KUKA KRL program: Rack_Verde_Cerrar_D.src, Rack_Verde_Cerrar_D.dat

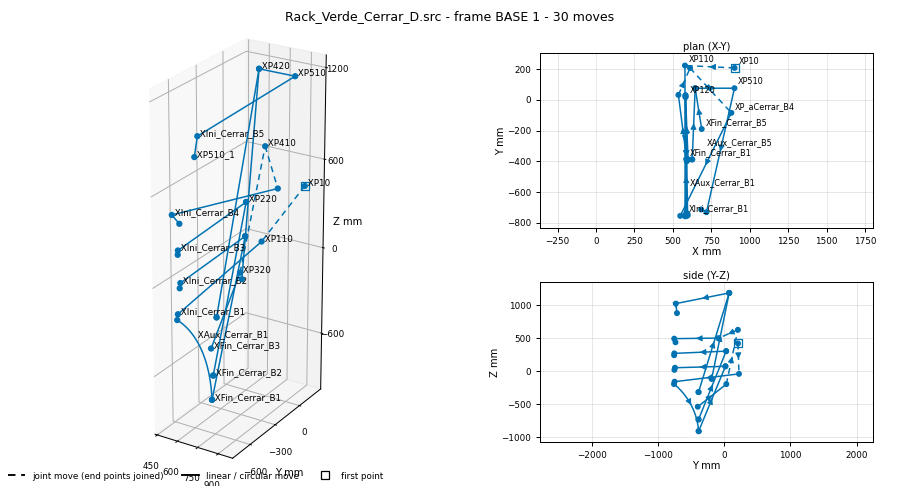
[picture p0: tool path of Rack_Verde_Cerrar_D.src in frame BASE 1, 30 of 38 moves have a stored position in this frame; points joined in program order, loops and branches not executed]
--- Rack_Verde_Cerrar_D.src ---
&ACCESS RVO1
&REL 165
&COMMENT CERRAR BANDEJAS PRG
&PARAM EDITMASK = *
&PARAM TEMPLATE = C:\KRC\Roboter\Template\vorgabe
&PARAM DISKPATH = KRC:\R1\Program\MAFELEC
DEF Rack_Verde_Cerrar_D( )
;FOLD INI;%{PE}
  ;FOLD BASISTECH INI
    GLOBAL INTERRUPT DECL 3 WHEN $STOPMESS==TRUE DO IR_STOPM ( )
    INTERRUPT ON 3
    BAS (#INITMOV,0 )
  ;ENDFOLD (BASISTECH INI)
;FOLD SPOTTECH INI
USERSPOT(#INIT)
;ENDFOLD (SPOTTECH INI)
;FOLD GRIPPERTECH INI
USER_GRP(0,DUMMY,DUMMY,GDEFAULT)
;ENDFOLD (GRIPPERTECH INI)
  ;FOLD USER INI
    ;Make your modifications here
INTERRUPT DECL 81 WHEN I_121R1S501 DO STOP_PUSH()
INTERRUPT DECL 91 WHEN I_121R1S502 DO STOP_PUSH()

O_TYPE_INFO=0

  ;ENDFOLD (USER INI)
;ENDFOLD (INI)
;################################################
; PROYECTO: MAFELEC PLANTA DE BATERIAS
; ROBOT: 121_R1
; PROGRAMA: CERRAR BANDEJAS EN RACK VERDE
; CREADO POR: Alejandro Company(zaisor robotics)
; FECHA: 23-NOVIEMBRE-2022
; MODIFICADO POR:
; FECHA MODIFICACION: 20-ENERO-2023
;################################################

$TIMER[5]=0
$TIMER_STOP[5]=FALSE

PTP $POS_ACT
Empujador(1,"A",FALSE)
Empujador(2,"R",FALSE)

;FOLD BORRADO SEÑALES INPICKER
O_INPICKER_OK=FALSE
O_INPICKER_NOK=FALSE
O_LIMITS_OK=FALSE
O_LIMITS_NOK=FALSE
O_LIMIT_X=FALSE
O_LIMIT_Y=FALSE
O_LIMIT_Z=FALSE
O_LIMIT_A=FALSE
O_LIMIT_B=FALSE
O_LIMIT_C=FALSE
;ENDFOLD

;INTERRUPT ON 81

INI_BUCLE:
;FOLD LIN P10 Vel=0.05 m/s M Tool[1]:T_PUSH1 Base[1]:Rack_Verde;%{PE}%R 8.3.48,%MKUKATPBASIS,%CMOVE,%VLIN,%P 1:LIN, 2:P10, 3:, 5:0.05, 7:M
$BWDSTART=FALSE
LDAT_ACT=LM
FDAT_ACT=FP10
BAS(#CP_PARAMS,0.05)
LIN XP10
;ENDFOLD

If ($SR_RANGE_ACTIVE[16]==FALSE) THEN
$out[61]=TRUE
WAIT FOR FALSE
WAIT FOR FALSE
WAIT FOR FALSE
;SETA DE BOMBEROS PULSADA, LLEVAR ROBOT A HOME Y REINICIAR PROGRAMA PARA RESTABLECER
ENDIF


WAIT FOR I_121R1S1000==FALSE
Empujador(1,"A",TRUE)
Empujador(2,"R",TRUE)
$ADVANCE=0

WAIT FOR (RV_Bandeja_Nr>10) AND (RV_Bandeja_Nr<16)

;PETICION CLAUSURA BANDEJAS EN RACK VERDE
SWITCH RV_Bandeja_Nr ;

CASE 11
O_TYPE_RQ=FALSE
O_TYPE_INFO=RV_Bandeja_Nr

;FOLD PTP P110 CONT Vel=50 % M Tool[1]:T_PUSH1 Base[1]:Rack_Verde;%{PE}%R 8.3.48,%MKUKATPBASIS,%CMOVE,%VPTP,%P 1:PTP, 2:P110, 3:C_DIS, 5:50, 7:M
$BWDSTART=FALSE
PDAT_ACT=PM
FDAT_ACT=FP110
BAS(#PTP_PARAMS,50)
PTP XP110 C_DIS
;ENDFOLD

WAIT FOR I_RackVerde_Pin1A
WAIT FOR I_Rack1_S1==TRUE
O_TREQ_2=TRUE

;FOLD LIN Ini_Cerrar_B1 Vel=1 m/s M Tool[1]:T_PUSH1 Base[1]:Rack_Verde;%{PE}%R 8.3.48,%MKUKATPBASIS,%CMOVE,%VLIN,%P 1:LIN, 2:Ini_Cerrar_B1, 3:, 5:1, 7:M
$BWDSTART=FALSE
LDAT_ACT=LM
FDAT_ACT=FIni_Cerrar_B1
BAS(#CP_PARAMS,1)
LIN XIni_Cerrar_B1
;ENDFOLD
;FOLD LIN P110_1 Vel=1 m/s M Tool[1]:T_PUSH1 Base[1]:Rack_Verde;%{PE}%R 8.3.48,%MKUKATPBASIS,%CMOVE,%VLIN,%P 1:LIN, 2:P110_1, 3:, 5:1, 7:M
$BWDSTART=FALSE
LDAT_ACT=LM
FDAT_ACT=FP110_1
BAS(#CP_PARAMS,1)
LIN XP110_1
;ENDFOLD

O_TREQ_2=TRUE
WAIT FOR I_TRDY_2
O_TREQ_2=FALSE

;FOLD CIRC Aux_Cerrar_B1 Fin_Cerrar_B1 Vel=1 m/s M Tool[1]:T_PUSH1 Base[1]:Rack_Verde;%{PE}%R 8.3.48,%MKUKATPBASIS,%CMOVE,%VCIRC,%P 1:CIRC, 2:Aux_Cerrar_B1, 3:Fin_Cerrar_B1, 4:, 6:1, 8:M
$BWDSTART=FALSE
LDAT_ACT=LM
FDAT_ACT=FFin_Cerrar_B1
BAS(#CP_PARAMS,1)
CIRC XAux_Cerrar_B1, XFin_Cerrar_B1
;ENDFOLD
;FOLD LIN Fin_Cerrar_B1 Vel=0.5 m/s CPDAT2 Tool[1]:T_PUSH1 Base[1]:Rack_Verde;%{PE}%R 8.3.48,%MKUKATPBASIS,%CMOVE,%VLIN,%P 1:LIN, 2:Fin_Cerrar_B1, 3:, 5:0.5, 7:CPDAT2
$BWDSTART=FALSE
LDAT_ACT=LCPDAT2
FDAT_ACT=FFin_Cerrar_B1
BAS(#CP_PARAMS,0.5)
LIN XFin_Cerrar_B1
;ENDFOLD
IF ($IN[64]==TRUE) THEN
;FOLD MOVIMIENTO CONTROLADO CERRAR BANDEJA

   $OUT[63]=TRUE ; DESHABILITAMOS EL CONTROL DE SOBREPASO EN PLC
   INTERRUPT OFF 81 ;DESHABILITAMOS LA INTERRUPCION
   Repite=0
   LIN_REL{Y 20}
   WHILE (I_121R1S501==FALSE) AND (Repite<=20);SENSOR SOBREPASO CLAMPA RACK AZUL

     Repite=Repite+1
     LIN_REL{Z -1}
     ;WAIT SEC 0.1

     ;IF Repite>=20 THEN
        ;HALT
         ;SUPERADO NUMERO DE REPETICIONES
        ;HALT
     ;ENDIF

   ENDWHILE


;ENDFOLD
ENDIF
;FOLD LIN P120 Vel=1 m/s M Tool[1]:T_PUSH1 Base[1]:Rack_Verde;%{PE}%R 8.3.48,%MKUKATPBASIS,%CMOVE,%VLIN,%P 1:LIN, 2:P120, 3:, 5:1, 7:M
$BWDSTART=FALSE
LDAT_ACT=LM
FDAT_ACT=FP120
BAS(#CP_PARAMS,1)
LIN XP120
;ENDFOLD

GOTO FIN

CASE 12

O_TYPE_RQ=FALSE
O_TYPE_INFO=RV_Bandeja_Nr

;FOLD PTP P210 CONT Vel=50 % M Tool[1]:T_PUSH1 Base[1]:Rack_Verde;%{PE}%R 8.3.48,%MKUKATPBASIS,%CMOVE,%VPTP,%P 1:PTP, 2:P210, 3:C_DIS, 5:50, 7:M
$BWDSTART=FALSE
PDAT_ACT=PM
FDAT_ACT=FP210
BAS(#PTP_PARAMS,50)
PTP XP210 C_DIS
;ENDFOLD

WAIT FOR I_RackVerde_Pin2A
WAIT FOR I_Rack1_S2==TRUE
WAIT FOR I_Rack1_S1==FALSE
O_TREQ_2=TRUE

;FOLD LIN Ini_Cerrar_B2 Vel=1 m/s M Tool[1]:T_PUSH1 Base[1]:Rack_Verde;%{PE}%R 8.3.48,%MKUKATPBASIS,%CMOVE,%VLIN,%P 1:LIN, 2:Ini_Cerrar_B2, 3:, 5:1, 7:M
$BWDSTART=FALSE
LDAT_ACT=LM
FDAT_ACT=FIni_Cerrar_B2
BAS(#CP_PARAMS,1)
LIN XIni_Cerrar_B2
;ENDFOLD
;FOLD LIN P210_1 Vel=1 m/s M Tool[1]:T_PUSH1 Base[1]:Rack_Verde;%{PE}%R 8.3.48,%MKUKATPBASIS,%CMOVE,%VLIN,%P 1:LIN, 2:P210_1, 3:, 5:1, 7:M
$BWDSTART=FALSE
LDAT_ACT=LM
FDAT_ACT=FP210_1
BAS(#CP_PARAMS,1)
LIN XP210_1
;ENDFOLD

O_TREQ_2=TRUE
WAIT FOR I_TRDY_2
O_TREQ_2=FALSE
PTP $POS_ACT

;FOLD CIRC Aux_Cerrar_B2 Fin_Cerrar_B2 Vel=1 m/s M Tool[1]:T_PUSH1 Base[1]:Rack_Verde;%{PE}%R 8.3.48,%MKUKATPBASIS,%CMOVE,%VCIRC,%P 1:CIRC, 2:Aux_Cerrar_B2, 3:Fin_Cerrar_B2, 4:, 6:1, 8:M
$BWDSTART=FALSE
LDAT_ACT=LM
FDAT_ACT=FFin_Cerrar_B2
BAS(#CP_PARAMS,1)
CIRC XAux_Cerrar_B2, XFin_Cerrar_B2
;ENDFOLD

;FOLD LIN Fin_Cerrar_B2 Vel=2 m/s M Tool[1]:T_PUSH1 Base[1]:Rack_Verde;%{PE}%R 8.3.48,%MKUKATPBASIS,%CMOVE,%VLIN,%P 1:LIN, 2:Fin_Cerrar_B2, 3:, 5:2, 7:M
$BWDSTART=FALSE
LDAT_ACT=LM
FDAT_ACT=FFin_Cerrar_B2
BAS(#CP_PARAMS,2)
LIN XFin_Cerrar_B2
;ENDFOLD
IF ($IN[64]==TRUE) THEN
;FOLD MOVIMIENTO CONTROLADO CERRAR BANDEJA

   $OUT[63]=TRUE ; DESHABILITAMOS EL CONTROL DE SOBREPASO EN PLC
   INTERRUPT OFF 81 ;DESHABILITAMOS LA INTERRUPCION
   Repite=0
   ;LIN_REL{Y 20}
   WHILE (I_121R1S501==FALSE) AND (Repite<=20);SENSOR SOBREPASO CLAMPA RACK AZUL

     Repite=Repite+1
     LIN_REL{Z -1}
     ;WAIT SEC 0.1

     ;IF Repite>=20 THEN
        ;HALT
         ;SUPERADO NUMERO DE REPETICIONES
        ;HALT
     ;ENDIF

   ENDWHILE


;ENDFOLD
ENDIF
;FOLD LIN P220 Vel=1 m/s M Tool[1]:T_PUSH1 Base[1]:Rack_Verde;%{PE}%R 8.3.48,%MKUKATPBASIS,%CMOVE,%VLIN,%P 1:LIN, 2:P220, 3:, 5:1, 7:M
$BWDSTART=FALSE
LDAT_ACT=LM
FDAT_ACT=FP220
BAS(#CP_PARAMS,1)
LIN XP220
;ENDFOLD

GOTO FIN

CASE 13
O_TYPE_RQ=FALSE
O_TYPE_INFO=RV_Bandeja_Nr

;FOLD LIN P310 CONT Vel=0.2 m/s L Tool[1]:T_PUSH1 Base[1]:Rack_Verde;%{PE}%R 8.3.48,%MKUKATPBASIS,%CMOVE,%VLIN,%P 1:LIN, 2:P310, 3:C_DIS C_DIS, 5:0.2, 7:L
$BWDSTART=FALSE
LDAT_ACT=LL
FDAT_ACT=FP310
BAS(#CP_PARAMS,0.2)
LIN XP310 C_DIS C_DIS
;ENDFOLD

WAIT FOR I_RackVerde_Pin3A
WAIT FOR I_Rack1_S3==TRUE
WAIT FOR I_Rack1_S2==FALSE
O_TREQ_2=TRUE

;FOLD LIN Ini_Cerrar_B3 Vel=1 m/s M Tool[1]:T_PUSH1 Base[1]:Rack_Verde;%{PE}%R 8.3.48,%MKUKATPBASIS,%CMOVE,%VLIN,%P 1:LIN, 2:Ini_Cerrar_B3, 3:, 5:1, 7:M
$BWDSTART=FALSE
LDAT_ACT=LM
FDAT_ACT=FIni_Cerrar_B3
BAS(#CP_PARAMS,1)
LIN XIni_Cerrar_B3
;ENDFOLD
;FOLD LIN P310_1 Vel=1 m/s M Tool[1]:T_PUSH1 Base[1]:Rack_Verde;%{PE}%R 8.3.48,%MKUKATPBASIS,%CMOVE,%VLIN,%P 1:LIN, 2:P310_1, 3:, 5:1, 7:M
$BWDSTART=FALSE
LDAT_ACT=LM
FDAT_ACT=FP310_1
BAS(#CP_PARAMS,1)
LIN XP310_1
;ENDFOLD

O_TREQ_2=TRUE
WAIT FOR I_TRDY_2
O_TREQ_2=FALSE
PTP $POS_ACT

;FOLD CIRC Aux_Cerrar_B3 Fin_Cerrar_B3 Vel=1 m/s M Tool[1]:T_PUSH1 Base[1]:Rack_Verde;%{PE}%R 8.3.48,%MKUKATPBASIS,%CMOVE,%VCIRC,%P 1:CIRC, 2:Aux_Cerrar_B3, 3:Fin_Cerrar_B3, 4:, 6:1, 8:M
$BWDSTART=FALSE
LDAT_ACT=LM
FDAT_ACT=FFin_Cerrar_B3
BAS(#CP_PARAMS,1)
CIRC XAux_Cerrar_B3, XFin_Cerrar_B3
;ENDFOLD
IF ($IN[64]==TRUE) THEN
;FOLD MOVIMIENTO CONTROLADO CERRAR BANDEJA

   $OUT[63]=TRUE ; DESHABILITAMOS EL CONTROL DE SOBREPASO EN PLC
   INTERRUPT OFF 81 ;DESHABILITAMOS LA INTERRUPCION
   Repite=0
   ;LIN_REL{Y 20}
   WHILE (I_121R1S501==FALSE) AND (Repite<=20);SENSOR SOBREPASO CLAMPA RACK AZUL

     Repite=Repite+1
     LIN_REL{Z -1}
     ;WAIT SEC 0.1

     ;IF Repite>=20 THEN
        ;HALT
         ;SUPERADO NUMERO DE REPETICIONES
        ;HALT
     ;ENDIF

   ENDWHILE


;ENDFOLD
ENDIF
;FOLD LIN P320 Vel=1 m/s M Tool[1]:T_PUSH1 Base[1]:Rack_Verde;%{PE}%R 8.3.48,%MKUKATPBASIS,%CMOVE,%VLIN,%P 1:LIN, 2:P320, 3:, 5:1, 7:M
$BWDSTART=FALSE
LDAT_ACT=LM
FDAT_ACT=FP320
BAS(#CP_PARAMS,1)
LIN XP320
;ENDFOLD

GOTO FIN

CASE 14
O_TYPE_RQ=FALSE
O_TYPE_INFO=RV_Bandeja_Nr

;FOLD PTP P410 CONT Vel=50 % M Tool[1]:T_PUSH1 Base[1]:Rack_Verde;%{PE}%R 8.3.48,%MKUKATPBASIS,%CMOVE,%VPTP,%P 1:PTP, 2:P410, 3:C_DIS, 5:50, 7:M
$BWDSTART=FALSE
PDAT_ACT=PM
FDAT_ACT=FP410
BAS(#PTP_PARAMS,50)
PTP XP410 C_DIS
;ENDFOLD

WAIT FOR I_RackVerde_Pin4A
WAIT FOR I_Rack1_S4==TRUE
WAIT FOR I_Rack1_S3==FALSE
O_TREQ_2=TRUE

;FOLD PTP P_aCerrar_B4 CONT Vel=50 % M Tool[1]:T_PUSH1 Base[1]:Rack_Verde;%{PE}%R 8.3.48,%MKUKATPBASIS,%CMOVE,%VPTP,%P 1:PTP, 2:P_aCerrar_B4, 3:C_DIS, 5:50, 7:M
$BWDSTART=FALSE
PDAT_ACT=PM
FDAT_ACT=FP_aCerrar_B4
BAS(#PTP_PARAMS,50)
PTP XP_aCerrar_B4 C_DIS
;ENDFOLD
;FOLD LIN Ini_Cerrar_B4 Vel=1 m/s M Tool[1]:T_PUSH1 Base[1]:Rack_Verde;%{PE}%R 8.3.48,%MKUKATPBASIS,%CMOVE,%VLIN,%P 1:LIN, 2:Ini_Cerrar_B4, 3:, 5:1, 7:M
$BWDSTART=FALSE
LDAT_ACT=LM
FDAT_ACT=FIni_Cerrar_B4
BAS(#CP_PARAMS,1)
LIN XIni_Cerrar_B4
;ENDFOLD

;FOLD LIN P410_1 Vel=1 m/s M Tool[1]:T_PUSH1 Base[1]:Rack_Verde;%{PE}%R 8.3.48,%MKUKATPBASIS,%CMOVE,%VLIN,%P 1:LIN, 2:P410_1, 3:, 5:1, 7:M
$BWDSTART=FALSE
LDAT_ACT=LM
FDAT_ACT=FP410_1
BAS(#CP_PARAMS,1)
LIN XP410_1
;ENDFOLD

O_TREQ_2=TRUE
WAIT FOR I_TRDY_2
O_TREQ_2=FALSE
PTP $POS_ACT

;FOLD CIRC Aux_Cerrar_B4 Fin_Cerrar_B4 Vel=1 m/s M Tool[1]:T_PUSH1 Base[1]:Rack_Verde;%{PE}%R 8.3.48,%MKUKATPBASIS,%CMOVE,%VCIRC,%P 1:CIRC, 2:Aux_Cerrar_B4, 3:Fin_Cerrar_B4, 4:, 6:1, 8:M
$BWDSTART=FALSE
LDAT_ACT=LM
FDAT_ACT=FFin_Cerrar_B4
BAS(#CP_PARAMS,1)
CIRC XAux_Cerrar_B4, XFin_Cerrar_B4
;ENDFOLD
;FOLD LIN Fin_Cerrar_B4 Vel=1 m/s M Tool[1]:T_PUSH1 Base[1]:Rack_Verde;%{PE}%R 8.3.48,%MKUKATPBASIS,%CMOVE,%VLIN,%P 1:LIN, 2:Fin_Cerrar_B4, 3:, 5:1, 7:M
$BWDSTART=FALSE
LDAT_ACT=LM
FDAT_ACT=FFin_Cerrar_B4
BAS(#CP_PARAMS,1)
LIN XFin_Cerrar_B4
;ENDFOLD
IF ($IN[64]==TRUE) THEN
;FOLD MOVIMIENTO CONTROLADO CERRAR BANDEJA

   $OUT[63]=TRUE ; DESHABILITAMOS EL CONTROL DE SOBREPASO EN PLC
   INTERRUPT OFF 81 ;DESHABILITAMOS LA INTERRUPCION
   Repite=0
   ;LIN_REL{Y 20}
   WHILE (I_121R1S501==FALSE) AND (Repite<=20);SENSOR SOBREPASO CLAMPA RACK AZUL

     Repite=Repite+1
     LIN_REL{Z -1}
     ;WAIT SEC 0.1

     ;IF Repite>=20 THEN
        ;HALT
         ;SUPERADO NUMERO DE REPETICIONES
        ;HALT
     ;ENDIF

   ENDWHILE


;ENDFOLD
ENDIF
;FOLD LIN P420 Vel=1 m/s M Tool[1]:T_PUSH1 Base[1]:Rack_Verde;%{PE}%R 8.3.48,%MKUKATPBASIS,%CMOVE,%VLIN,%P 1:LIN, 2:P420, 3:, 5:1, 7:M
$BWDSTART=FALSE
LDAT_ACT=LM
FDAT_ACT=FP420
BAS(#CP_PARAMS,1)
LIN XP420
;ENDFOLD

GOTO FIN

CASE 15
O_TYPE_RQ=FALSE
O_TYPE_INFO=RV_Bandeja_Nr

;FOLD LIN P510 CONT Vel=1 m/s M Tool[1]:T_PUSH1 Base[1]:Rack_Verde;%{PE}%R 8.3.48,%MKUKATPBASIS,%CMOVE,%VLIN,%P 1:LIN, 2:P510, 3:C_DIS C_DIS, 5:1, 7:M
$BWDSTART=FALSE
LDAT_ACT=LM
FDAT_ACT=FP510
BAS(#CP_PARAMS,1)
LIN XP510 C_DIS C_DIS
;ENDFOLD

WAIT FOR I_RackVerde_Pin5A
WAIT FOR I_Rack1_S5==TRUE
WAIT FOR I_Rack1_S4==FALSE
O_TREQ_2=TRUE

;FOLD LIN Ini_Cerrar_B5 Vel=1 m/s M Tool[1]:T_PUSH1 Base[1]:Rack_Verde;%{PE}%R 8.3.48,%MKUKATPBASIS,%CMOVE,%VLIN,%P 1:LIN, 2:Ini_Cerrar_B5, 3:, 5:1, 7:M
$BWDSTART=FALSE
LDAT_ACT=LM
FDAT_ACT=FIni_Cerrar_B5
BAS(#CP_PARAMS,1)
LIN XIni_Cerrar_B5
;ENDFOLD

;FOLD LIN P510_1 Vel=1 m/s M Tool[1]:T_PUSH1 Base[1]:Rack_Verde;%{PE}%R 8.3.48,%MKUKATPBASIS,%CMOVE,%VLIN,%P 1:LIN, 2:P510_1, 3:, 5:1, 7:M
$BWDSTART=FALSE
LDAT_ACT=LM
FDAT_ACT=FP510_1
BAS(#CP_PARAMS,1)
LIN XP510_1
;ENDFOLD

O_TREQ_2=TRUE
WAIT FOR I_TRDY_2
O_TREQ_2=FALSE
PTP $POS_ACT

;FOLD CIRC Aux_Cerrar_B5 Fin_Cerrar_B5 Vel=1 m/s M Tool[1]:T_PUSH1 Base[1]:Rack_Verde;%{PE}%R 8.3.48,%MKUKATPBASIS,%CMOVE,%VCIRC,%P 1:CIRC, 2:Aux_Cerrar_B5, 3:Fin_Cerrar_B5, 4:, 6:1, 8:M
$BWDSTART=FALSE
LDAT_ACT=LM
FDAT_ACT=FFin_Cerrar_B5
BAS(#CP_PARAMS,1)
CIRC XAux_Cerrar_B5, XFin_Cerrar_B5
;ENDFOLD
IF ($IN[64]==TRUE) THEN
;FOLD MOVIMIENTO CONTROLADO CERRAR BANDEJA

   $OUT[63]=TRUE ; DESHABILITAMOS EL CONTROL DE SOBREPASO EN PLC
   INTERRUPT OFF 81 ;DESHABILITAMOS LA INTERRUPCION
   Repite=0
   ;LIN_REL{Y 20}
   WHILE (I_121R1S501==FALSE) AND (Repite<=20);SENSOR SOBREPASO CLAMPA RACK AZUL

     Repite=Repite+1
     LIN_REL{Z -1}
     ;WAIT SEC 0.1

     ;IF Repite>=20 THEN
        ;HALT
         ;SUPERADO NUMERO DE REPETICIONES
        ;HALT
     ;ENDIF

   ENDWHILE


;ENDFOLD
ENDIF
;FOLD LIN P520 Vel=1 m/s M Tool[1]:T_PUSH1 Base[1]:Rack_Verde;%{PE}%R 8.3.48,%MKUKATPBASIS,%CMOVE,%VLIN,%P 1:LIN, 2:P520, 3:, 5:1, 7:M
$BWDSTART=FALSE
LDAT_ACT=LM
FDAT_ACT=FP520
BAS(#CP_PARAMS,1)
LIN XP520
;ENDFOLD

GOTO FIN

DEFAULT
HALT
HALT
; #### CODIGO ERRONEO ####
HALT
BRAKE

ENDSWITCH

FIN:

$ADVANCE=3

; POSICION DE SALIDA RACK 1
;FOLD PTP POS_AREA1_LIBRE Vel=100 % H Tool[9]:T_Gripper1_Vacio Base[0];%{PE}%R 8.3.48,%MKUKATPBASIS,%CMOVE,%VPTP,%P 1:PTP, 2:POS_AREA1_LIBRE, 3:, 5:100, 7:H
$BWDSTART=FALSE
PDAT_ACT=PH
FDAT_ACT=FPOS_AREA1_LIBRE
BAS(#PTP_PARAMS,100)
PTP XPOS_AREA1_LIBRE
;ENDFOLD

; TRABAJO REALIZADO
O_JRDY_4=TRUE

Empujador(1,"R",FALSE)
Empujador(2,"R",FALSE)

O_AREL_1=TRUE

;FOLD PTP P_aHOME CONT Vel=100 % H Tool[9]:T_Gripper1_Vacio Base[0];%{PE}%R 8.3.48,%MKUKATPBASIS,%CMOVE,%VPTP,%P 1:PTP, 2:P_aHOME, 3:C_DIS, 5:100, 7:H
$BWDSTART=FALSE
PDAT_ACT=PH
FDAT_ACT=FP_aHOME
BAS(#PTP_PARAMS,100)
PTP XP_aHOME C_DIS
;ENDFOLD

Empujador(1,"R",TRUE)
Empujador(2,"R",TRUE)

$TIMER_STOP[5]=TRUE
END
DEF STOP_PUSH()
INTERRUPT OFF 81

IF $PRO_MOVE THEN

BRAKE

IF NOT $ON_PATH THEN
PTP $AXIS_ACT
ENDIF

ENDIF

LIN_REL{Z +50}
WAIT FOR (NOT I_121R1S501) AND (NOT I_121R1S502)

INTERRUPT ON 81
END

--- Rack_Verde_Cerrar_D.dat ---
&ACCESS RVO1
&REL 165
&COMMENT CERRAR BANDEJAS PRG
&PARAM EDITMASK = *
&PARAM TEMPLATE = C:\KRC\Roboter\Template\vorgabe
&PARAM DISKPATH = KRC:\R1\Program\MAFELEC
DEFDAT  Rack_Verde_Cerrar_D
;FOLD EXTERNAL DECLARATIONS;%{PE}%MKUKATPBASIS,%CEXT,%VCOMMON,%P
;FOLD GRIPPERTECH EXT
EXT  H50 (INT  :IN,INT  :IN,INT  :IN,GRP_TYP  :IN )
;ENDFOLD (GRIPPERTECH EXT)
;FOLD SPOTTECH EXT
EXT  USERSPOT (S_COMMAND  :IN,SPOT_TYPE  :IN )
;ENDFOLD (SPOTTECH EXT)
;FOLD BASISTECH EXT;%{PE}%MKUKATPBASIS,%CEXT,%VEXT,%P
EXT  BAS (BAS_COMMAND  :IN,REAL  :IN )
DECL INT SUCCESS
;ENDFOLD (BASISTECH EXT)
;FOLD USER EXT;%{E}%MKUKATPUSER,%CEXT,%VEXT,%P
;Make your modifications here

;ENDFOLD (USER EXT)
;ENDFOLD (EXTERNAL DECLARATIONS)
DECL BASIS_SUGG_T LAST_BASIS={POINT1[] "P0                      ",POINT2[] "P0                      ",CP_PARAMS[] "CPDAT0                  ",PTP_PARAMS[] "PDAT0                   ",CONT[] "                        ",CP_VEL[] "0.05                    ",PTP_VEL[] "100                     ",SYNC_PARAMS[] "SYNCDAT                 ",SPL_NAME[] "S0                      ",A_PARAMS[] "ADAT0                   "}
DECL PDAT PH={VEL 100.000,ACC 100.000,APO_DIST 100.000,APO_MODE #CDIS,GEAR_JERK 50.0000,EXAX_IGN 0}
DECL E6POS XPOS_ESPERA_AREA1={X 112.943756,Y -227.851166,Z 2716.11304,A 36.2463837,B -15.5853510,C 56.0520973,S 3,T 42,E1 0.0,E2 0.0,E3 0.0,E4 0.0,E5 0.0,E6 0.0}
DECL FDAT FPOS_ESPERA_AREA1={TOOL_NO 9,BASE_NO 0,IPO_FRAME #BASE,POINT2[] " ",TQ_STATE FALSE}
DECL LDAT LL={VEL 2.00000,ACC 15.0000,APO_DIST 40.0000,APO_FAC 50.0000,AXIS_VEL 100.000,AXIS_ACC 100.000,ORI_TYP #VAR,CIRC_TYP #BASE,JERK_FAC 50.0000,GEAR_JERK 50.0000,EXAX_IGN 0}
DECL E6POS XPOS_AREA1_LIBRE={X -250.533554,Y -43.6507149,Z 2716.11304,A -84.6604385,B 6.50295877,C 57.2217522,S 3,T 42,E1 0.0,E2 0.0,E3 0.0,E4 0.0,E5 0.0,E6 0.0}
DECL FDAT FPOS_AREA1_LIBRE={TOOL_NO 9,BASE_NO 0,IPO_FRAME #BASE,POINT2[] " ",TQ_STATE FALSE}
DECL E6POS XP111={X 557.799622,Y -753.947571,Z -222.785736,A -88.9974060,B 13.7721291,C 89.1738281,S 6,T 58,E1 0.0,E2 0.0,E3 0.0,E4 0.0,E5 0.0,E6 0.0}
DECL FDAT FP111={TOOL_NO 1,BASE_NO 1,IPO_FRAME #BASE,POINT2[] " ",TQ_STATE FALSE}
DECL E6POS XP10={X 901.450,Y 208.526413,Z 420.362366,A -90.0963,B 3.32343674,C 88.1521912,S 2,T 34,E1 0.0,E2 0.0,E3 0.0,E4 0.0,E5 0.0,E6 0.0}
DECL FDAT FP10={TOOL_NO 1,BASE_NO 1,IPO_FRAME #BASE,POINT2[] " ",TQ_STATE FALSE}
DECL E6POS XP110={X 578.741150,Y 224.019104,Z -39.7154198,A -89.1475,B 1.10093117,C 89.1576843,S 6,T 50,E1 0.0,E2 0.0,E3 0.0,E4 0.0,E5 0.0,E6 0.0}
DECL FDAT FP110={TOOL_NO 1,BASE_NO 1,IPO_FRAME #BASE,POINT2[] " ",TQ_STATE FALSE}
DECL E6POS XP120={X 582.226318,Y 19.1561737,Z 74.4672852,A -88.9195404,B 4.33784628,C 89.1742401,S 6,T 58,E1 0.0,E2 0.0,E3 0.0,E4 0.0,E5 0.0,E6 0.0}
DECL FDAT FP120={TOOL_NO 1,BASE_NO 1,IPO_FRAME #BASE,POINT2[] " ",TQ_STATE FALSE}
DECL E6POS XP_ABRIR10={X -250.533554,Y -43.6507149,Z 2716.11304,A -84.6604385,B 6.50295877,C 57.2217522,S 3,T 42,E1 0.0,E2 0.0,E3 0.0,E4 0.0,E5 0.0,E6 0.0}
DECL FDAT FP_ABRIR10={TOOL_NO 9,BASE_NO 0,IPO_FRAME #BASE,POINT2[] " ",TQ_STATE FALSE}
DECL E6POS XP_AHOME={X 112.943756,Y -227.851166,Z 2716.11304,A 36.2463837,B -15.5853510,C 56.0520973,S 3,T 42,E1 0.0,E2 0.0,E3 0.0,E4 0.0,E5 0.0,E6 0.0}
DECL FDAT FP_aHOME={TOOL_NO 9,BASE_NO 0,IPO_FRAME #BASE,POINT2[] " ",TQ_STATE FALSE}
DECL E6POS XIni_Cerrar_B1={X 579.364929,Y -748.520142,Z -157.430450,A -89.0192184,B 10.1963968,C 89.1201324,S 6,T 58,E1 0.0,E2 0.0,E3 0.0,E4 0.0,E5 0.0,E6 0.0}
DECL FDAT FIni_Cerrar_B1={TOOL_NO 1,BASE_NO 1,IPO_FRAME #BASE,POINT2[] " ",TQ_STATE FALSE}
DECL E6POS XAux_Cerrar_B1={X 585.738403,Y -577.253296,Z -382.951569,A -88.8921585,B 21.8754425,C 89.7166061,S 6,T 58,E1 0.0,E2 0.0,E3 0.0,E4 0.0,E5 0.0,E6 0.0}
DECL E6POS XFin_Cerrar_B1={X 587.709595,Y -384.925323,Z -905.012939,A -88.0520859,B 34.1012230,C 90.8551254,S 6,T 58,E1 0.0,E2 0.0,E3 0.0,E4 0.0,E5 0.0,E6 0.0}
DECL FDAT FFin_Cerrar_B1={TOOL_NO 1,BASE_NO 1,IPO_FRAME #BASE,POINT2[] " ",TQ_STATE FALSE}
DECL E6POS XP0={X 632.645691,Y 303.475861,Z -186.174820,A -88.8950272,B 31.1322117,C 89.5053635,S 6,T 58,E1 0.0,E2 0.0,E3 0.0,E4 0.0,E5 0.0,E6 0.0}
DECL FDAT FP0={TOOL_NO 1,BASE_NO 1,IPO_FRAME #BASE,POINT2[] " ",TQ_STATE FALSE}
DECL E6POS XIni_Cerrar_B2={X 596.015869,Y -742.491516,Z 53.0099831,A -89.4107361,B 1.91299403,C 90.2672882,S 6,T 58,E1 0.0,E2 0.0,E3 0.0,E4 0.0,E5 0.0,E6 0.0}
DECL FDAT FIni_Cerrar_B2={TOOL_NO 1,BASE_NO 1,IPO_FRAME #BASE,POINT2[] " ",TQ_STATE FALSE}
DECL E6POS XP1={X 633.606323,Y -740.251,Z -11.7250,A -89.0051498,B 9.17837143,C 89.0890656,S 6,T 58,E1 0.0,E2 0.0,E3 0.0,E4 0.0,E5 0.0,E6 0.0}
DECL FDAT FP1={TOOL_NO 1,BASE_NO 1,IPO_FRAME #BASE,POINT2[] " ",TQ_STATE FALSE}
DECL E6POS XAux_Cerrar_B2={X 600.454773,Y -593.703735,Z -155.772568,A -89.5594330,B 18.2327461,C 90.1700592,S 6,T 58,E1 0.0,E2 0.0,E3 0.0,E4 0.0,E5 0.0,E6 0.0}
DECL E6POS XFin_Cerrar_B2={X 598.907471,Y -386.855804,Z -728.041809,A -90.0763397,B 33.4312744,C 89.5435791,S 6,T 58,E1 0.0,E2 0.0,E3 0.0,E4 0.0,E5 0.0,E6 0.0}
DECL FDAT FFin_Cerrar_B2={TOOL_NO 1,BASE_NO 1,IPO_FRAME #BASE,POINT2[] " ",TQ_STATE FALSE}
DECL E6POS XP2={X 535.775818,Y 225.276917,Z -536.621948,A -91.0083771,B 14.9493265,C 94.2730637,S 6,T 58,E1 0.0,E2 0.0,E3 0.0,E4 0.0,E5 0.0,E6 0.0}
DECL FDAT FP2={TOOL_NO 1,BASE_NO 1,IPO_FRAME #BASE,POINT2[] " ",TQ_STATE FALSE}
DECL E6POS XP210={X 582.226318,Y 19.1561737,Z 74.4672852,A -88.9195404,B 4.33784628,C 89.1742401,S 6,T 58,E1 0.0,E2 0.0,E3 0.0,E4 0.0,E5 0.0,E6 0.0}
DECL FDAT FP210={TOOL_NO 1,BASE_NO 1,IPO_FRAME #BASE,POINT2[] " ",TQ_STATE FALSE}
DECL E6POS XP220={X 582.225220,Y 30.3758373,Z 303.796967,A -88.9226303,B 4.33638334,C 89.1649170,S 6,T 58,E1 0.0,E2 0.0,E3 0.0,E4 0.0,E5 0.0,E6 0.0}
DECL FDAT FP220={TOOL_NO 1,BASE_NO 1,IPO_FRAME #BASE,POINT2[] " ",TQ_STATE FALSE}
DECL E6POS XP3={X 536.241516,Y 225.176605,Z 24.6719704,A -90.9851761,B 14.9447651,C 94.2668762,S 6,T 58,E1 0.0,E2 0.0,E3 0.0,E4 0.0,E5 0.0,E6 0.0}
DECL FDAT FP3={TOOL_NO 1,BASE_NO 1,IPO_FRAME #BASE,POINT2[] " ",TQ_STATE FALSE}
DECL E6POS XIni_Cerrar_B3={X 587.541870,Y -752.408,Z 269.800476,A -90.7068863,B 4.83034372,C 89.8440933,S 2,T 34,E1 0.0,E2 0.0,E3 0.0,E4 0.0,E5 0.0,E6 0.0}
DECL FDAT FIni_Cerrar_B3={TOOL_NO 1,BASE_NO 1,IPO_FRAME #BASE,POINT2[] " ",TQ_STATE FALSE}
DECL E6POS XP4={X 633.606323,Y -740.251,Z -11.7250,A -89.0051498,B 9.17837143,C 89.0890656,S 6,T 58,E1 0.0,E2 0.0,E3 0.0,E4 0.0,E5 0.0,E6 0.0}
DECL FDAT FP4={TOOL_NO 1,BASE_NO 1,IPO_FRAME #BASE,POINT2[] " ",TQ_STATE FALSE}
DECL E6POS XAux_Cerrar_B3={X 588.440369,Y -562.772644,Z 14.7120342,A -90.4545898,B 19.0679455,C 90.3643723,S 2,T 34,E1 0.0,E2 0.0,E3 0.0,E4 0.0,E5 0.0,E6 0.0}
DECL E6POS XFin_Cerrar_B3={X 591.055359,Y -398.157593,Z -535.615051,A -90.0148697,B 32.9485512,C 91.9439316,S 2,T 34,E1 0.0,E2 0.0,E3 0.0,E4 0.0,E5 0.0,E6 0.0}
DECL FDAT FFin_Cerrar_B3={TOOL_NO 1,BASE_NO 1,IPO_FRAME #BASE,POINT2[] "XAux_Cerrar_B3",TQ_STATE FALSE}
DECL E6POS XP5={X 535.775818,Y 225.276917,Z -194.099075,A -91.0083771,B 14.9493265,C 94.2730637,S 6,T 58,E1 0.0,E2 0.0,E3 0.0,E4 0.0,E5 0.0,E6 0.0}
DECL FDAT FP5={TOOL_NO 1,BASE_NO 1,IPO_FRAME #BASE,POINT2[] " ",TQ_STATE FALSE}
DECL E6POS XP310={X 582.225220,Y 30.3758373,Z 303.796967,A -88.9226303,B 4.33638334,C 89.1649170,S 6,T 58,E1 0.0,E2 0.0,E3 0.0,E4 0.0,E5 0.0,E6 0.0}
DECL FDAT FP310={TOOL_NO 1,BASE_NO 1,IPO_FRAME #BASE,POINT2[] " ",TQ_STATE FALSE}
DECL E6POS XP320={X 536.044250,Y 32.8823090,Z -194.276825,A -91.0112381,B 14.9554100,C 94.2986832,S 6,T 58,E1 0.0,E2 0.0,E3 0.0,E4 0.0,E5 0.0,E6 0.0}
DECL FDAT FP320={TOOL_NO 1,BASE_NO 1,IPO_FRAME #BASE,POINT2[] " ",TQ_STATE FALSE}
DECL E6POS XP310_1={X 587.542603,Y -754.938782,Z 242.364258,A -90.7068863,B 4.83034372,C 89.8440933,S 2,T 34,E1 0.0,E2 0.0,E3 0.0,E4 0.0,E5 0.0,E6 0.0}
DECL FDAT FP310_1={TOOL_NO 1,BASE_NO 1,IPO_FRAME #BASE,POINT2[] " ",TQ_STATE FALSE}
DECL E6POS XP6={X 536.241516,Y 225.176605,Z 24.6719704,A -90.9851761,B 14.9447651,C 94.2668762,S 6,T 58,E1 0.0,E2 0.0,E3 0.0,E4 0.0,E5 0.0,E6 0.0}
DECL FDAT FP6={TOOL_NO 1,BASE_NO 1,IPO_FRAME #BASE,POINT2[] " ",TQ_STATE FALSE}
DECL E6POS XIni_Cerrar_B4={X 547.969421,Y -753.810364,Z 492.527710,A -91.9702,B 13.7009811,C 90.2765808,S 6,T 26,E1 0.0,E2 0.0,E3 0.0,E4 0.0,E5 0.0,E6 0.0}
DECL FDAT FIni_Cerrar_B4={TOOL_NO 1,BASE_NO 1,IPO_FRAME #BASE,POINT2[] " ",TQ_STATE FALSE}
DECL E6POS XP7={X 633.606323,Y -740.251,Z -11.7250,A -89.0051498,B 9.17837143,C 89.0890656,S 6,T 58,E1 0.0,E2 0.0,E3 0.0,E4 0.0,E5 0.0,E6 0.0}
DECL FDAT FP7={TOOL_NO 1,BASE_NO 1,IPO_FRAME #BASE,POINT2[] " ",TQ_STATE FALSE}
DECL E6POS XAux_Cerrar_B4={X 590.257263,Y -584.788818,Z 231.681229,A -92.0750122,B 23.8326550,C 90.1046524,S 6,T 26,E1 0.0,E2 0.0,E3 0.0,E4 0.0,E5 0.0,E6 0.0}
DECL E6POS XFin_Cerrar_B4={X 625.953369,Y -386.815704,Z -314.899353,A -92.0722809,B 25.1516895,C 90.1206894,S 6,T 58,E1 0.0,E2 0.0,E3 0.0,E4 0.0,E5 0.0,E6 0.0}
DECL FDAT FFin_Cerrar_B4={TOOL_NO 1,BASE_NO 1,IPO_FRAME #BASE,POINT2[] " ",TQ_STATE FALSE}
DECL E6POS XP8={X 535.775818,Y 225.276917,Z -194.099075,A -91.0083771,B 14.9493265,C 94.2730637,S 6,T 58,E1 0.0,E2 0.0,E3 0.0,E4 0.0,E5 0.0,E6 0.0}
DECL FDAT FP8={TOOL_NO 1,BASE_NO 1,IPO_FRAME #BASE,POINT2[] " ",TQ_STATE FALSE}
DECL E6POS XP410={X 611.764221,Y 207.452301,Z 625.488281,A -86.7999649,B -2.01266837,C 87.2028,S 6,T 50,E1 0.0,E2 0.0,E3 0.0,E4 0.0,E5 0.0,E6 0.0}
DECL FDAT FP410={TOOL_NO 1,BASE_NO 1,IPO_FRAME #BASE,POINT2[] " ",TQ_STATE FALSE}
DECL E6POS XP410_1={X 588.247,Y -734.354614,Z 437.282227,A -92.0155411,B 18.5575695,C 90.2621613,S 6,T 26,E1 0.0,E2 0.0,E3 0.0,E4 0.0,E5 0.0,E6 0.0}
DECL FDAT FP410_1={TOOL_NO 1,BASE_NO 1,IPO_FRAME #BASE,POINT2[] " ",TQ_STATE FALSE}
DECL E6POS XP420={X 645.022156,Y 76.2896881,Z 1182.24231,A -101.552437,B 3.47349191,C 81.6571579,S 6,T 26,E1 0.0,E2 0.0,E3 0.0,E4 0.0,E5 0.0,E6 0.0}
DECL FDAT FP420={TOOL_NO 1,BASE_NO 1,IPO_FRAME #BASE,POINT2[] " ",TQ_STATE FALSE}
DECL E6POS XP9={X 536.241516,Y 225.176605,Z 24.6719704,A -90.9851761,B 14.9447651,C 94.2668762,S 6,T 58,E1 0.0,E2 0.0,E3 0.0,E4 0.0,E5 0.0,E6 0.0}
DECL FDAT FP9={TOOL_NO 1,BASE_NO 1,IPO_FRAME #BASE,POINT2[] " ",TQ_STATE FALSE}
DECL E6POS XIni_Cerrar_B5={X 718.579712,Y -729.796204,Z 1021.40900,A -90.2056,B 8.16238,C 88.6756210,S 6,T 26,E1 0.0,E2 0.0,E3 0.0,E4 0.0,E5 0.0,E6 0.0}
DECL FDAT FIni_Cerrar_B5={TOOL_NO 1,BASE_NO 1,IPO_FRAME #BASE,POINT2[] " ",TQ_STATE FALSE}
DECL E6POS XP11={X 633.606323,Y -740.251,Z -11.7250,A -89.0051498,B 9.17837143,C 89.0890656,S 6,T 58,E1 0.0,E2 0.0,E3 0.0,E4 0.0,E5 0.0,E6 0.0}
DECL FDAT FP11={TOOL_NO 1,BASE_NO 1,IPO_FRAME #BASE,POINT2[] " ",TQ_STATE FALSE}
DECL E6POS XAux_Cerrar_B5={X 693.645081,Y -318.877411,Z 443.374756,A -88.7919769,B 13.6895771,C 89.2889252,S 2,T 34,E1 0.0,E2 0.0,E3 0.0,E4 0.0,E5 0.0,E6 0.0}
DECL E6POS XFin_Cerrar_B5={X 687.616821,Y -188.913666,Z -116.045700,A -87.1484451,B 19.2286301,C 90.2566376,S 2,T 34,E1 0.0,E2 0.0,E3 0.0,E4 0.0,E5 0.0,E6 0.0}
DECL FDAT FFin_Cerrar_B5={TOOL_NO 1,BASE_NO 1,IPO_FRAME #BASE,POINT2[] "XAux_Cerrar_B5",TQ_STATE FALSE}
DECL E6POS XP12={X 535.775818,Y 225.276917,Z -194.099075,A -91.0083771,B 14.9493265,C 94.2730637,S 6,T 58,E1 0.0,E2 0.0,E3 0.0,E4 0.0,E5 0.0,E6 0.0}
DECL FDAT FP12={TOOL_NO 1,BASE_NO 1,IPO_FRAME #BASE,POINT2[] " ",TQ_STATE FALSE}
DECL E6POS XP510={X 900.618286,Y 76.5303802,Z 1182.48596,A -90.1547470,B 3.31829572,C 88.1377945,S 2,T 34,E1 0.0,E2 0.0,E3 0.0,E4 0.0,E5 0.0,E6 0.0}
DECL FDAT FP510={TOOL_NO 1,BASE_NO 1,IPO_FRAME #BASE,POINT2[] " ",TQ_STATE FALSE}
DECL E6POS XP510_1={X 684.525085,Y -712.085327,Z 877.389343,A -90.4030838,B 16.3972168,C 88.6339188,S 2,T 34,E1 0.0,E2 0.0,E3 0.0,E4 0.0,E5 0.0,E6 0.0}
DECL FDAT FP510_1={TOOL_NO 1,BASE_NO 1,IPO_FRAME #BASE,POINT2[] " ",TQ_STATE FALSE}
DECL E6POS XP520={X 645.022156,Y 76.2896881,Z 1182.24231,A -101.552437,B 3.47349191,C 81.6571579,S 6,T 26,E1 0.0,E2 0.0,E3 0.0,E4 0.0,E5 0.0,E6 0.0}
DECL FDAT FP520={TOOL_NO 1,BASE_NO 1,IPO_FRAME #BASE,POINT2[] " ",TQ_STATE FALSE}
DECL E6POS XP210_1={X 596.198059,Y -750.991699,Z 21.4653397,A -89.3987198,B 8.08528328,C 90.3318939,S 6,T 58,E1 0.0,E2 0.0,E3 0.0,E4 0.0,E5 0.0,E6 0.0}
DECL FDAT FP210_1={TOOL_NO 1,BASE_NO 1,IPO_FRAME #BASE,POINT2[] " ",TQ_STATE FALSE}
DECL E6POS XP110_1={X 579.443115,Y -756.902832,Z -193.088074,A -89.3051376,B 10.6269426,C 89.1188660,S 6,T 58,E1 0.0,E2 0.0,E3 0.0,E4 0.0,E5 0.0,E6 0.0}
DECL FDAT FP110_1={TOOL_NO 1,BASE_NO 1,IPO_FRAME #BASE,POINT2[] " ",TQ_STATE FALSE}
DECL E6POS XP_FIN={X 901.450,Y 208.526413,Z 420.362366,A -90.0963,B 3.32343674,C 88.1521912,S 6,T 26,E1 0.0,E2 0.0,E3 0.0,E4 0.0,E5 0.0,E6 0.0}
DECL FDAT FP_FIN={TOOL_NO 1,BASE_NO 1,IPO_FRAME #BASE,POINT2[] " ",TQ_STATE FALSE}
DECL E6POS XPCONEX={X 850.773865,Y 724.424316,Z 273.456970,A -87.1000290,B -0.167936072,C 179.536102,S 2,T 42,E1 0.0,E2 0.0,E3 0.0,E4 0.0,E5 0.0,E6 0.0}
DECL FDAT FPCONEX={TOOL_NO 9,BASE_NO 1,IPO_FRAME #BASE,POINT2[] " ",TQ_STATE FALSE}
DECL PDAT PPDAT1={VEL 100.000,ACC 100.000,APO_DIST 100.000,GEAR_JERK 50.0000,EXAX_IGN 0}
DECL PDAT PM={VEL 100.000,ACC 50.0000,APO_DIST 100.000,APO_MODE #CDIS,GEAR_JERK 50.0000,EXAX_IGN 0}
DECL E6POS XP_ACERRAR_B4={X 880.512878,Y -83.8103714,Z 500.720398,A -77.0251770,B 3.69670939,C 72.7839661,S 6,T 58,E1 0.0,E2 0.0,E3 0.0,E4 0.0,E5 0.0,E6 0.0}
DECL FDAT FP_aCerrar_B4={TOOL_NO 1,BASE_NO 1,IPO_FRAME #BASE,POINT2[] " ",TQ_STATE FALSE}
DECL LDAT LM={VEL 2.00000,ACC 25.0000,APO_DIST 100.000,APO_FAC 50.0000,AXIS_VEL 100.000,AXIS_ACC 100.000,ORI_TYP #VAR,CIRC_TYP #BASE,JERK_FAC 50.0000,GEAR_JERK 50.0000,EXAX_IGN 0}
DECL PDAT PPDAT2={VEL 100.000,ACC 50.0000,APO_DIST 100.000,APO_MODE #CDIS,GEAR_JERK 50.0000,EXAX_IGN 0}
DECL LDAT LCPDAT1={VEL 2.00000,ACC 10.0000,APO_DIST 100.000,APO_FAC 50.0000,AXIS_VEL 100.000,AXIS_ACC 100.000,ORI_TYP #VAR,CIRC_TYP #BASE,JERK_FAC 50.0000,GEAR_JERK 50.0000,EXAX_IGN 0}
DECL PDAT PPDAT3={VEL 100.000,ACC 50.0000,APO_DIST 100.000,GEAR_JERK 50.0000,EXAX_IGN 0}
DECL LDAT LCPDAT2={VEL 2.00000,ACC 25.0000,APO_DIST 100.000,APO_FAC 50.0000,AXIS_VEL 100.000,AXIS_ACC 100.000,ORI_TYP #VAR,CIRC_TYP #BASE,JERK_FAC 50.0000,GEAR_JERK 50.0000,EXAX_IGN 0}
ENDDAT
